PROGRAM MAIN
VAR
	State: INT;
	XtsMoverFactory : MoverFactory;
	XtsStationFactory : StationFactory;
	XtsTrackFactory : TrackFactory;
	iFactory : ITF_Factory := XtsMoverFactory;
	XtsElements : ARRAY[0..8] OF ITF_Cyclic;
	
	iMover : ITF_Mover;
	MaxVelo : LREAL;
	xTest: BOOL;
END_VAR

CASE State OF
	0:
		IF Initialise() THEN
			State := 1;
		END_IF
END_CASE

IF xTest THEN
	xTest := FALSE;
	IF __QUERYINTERFACE(XtsElements[1],iMover) THEN
		MaxVelo := iMover.GetMaxVelo();
	END_IF
END_IF

METHOD Initialise : BOOL
VAR_INPUT
END_VAR

VAR
	i: INT;
END_VAR
FOR i := 0 TO 2 DO
	XtsElements[i] := iFactory.Create();
END_FOR
iFactory := XtsStationFactory;
FOR i := 3 TO 5 DO
	XtsElements[i] := iFactory.Create();
END_FOR
iFactory := XtsTrackFactory;
FOR i := 6 TO 8 DO
	XtsElements[i] := iFactory.Create();
END_FOR
Initialise := TRUE;
END_METHOD

END_PROGRAM

(* stored: Version 1.1.0.1, ProductVersion 3.1.4024.12
   POU MAIN: Id {3dd2c997-63f0-4cd6-a20a-d17b2f2e0506}, SpecialFunc None
   Method Initialise: Id {97f2d371-0746-4166-ae23-b80a4f13a3c7} *)
